# EPICS substitutions: splineApp/Db/transformations.substitutions
file spline.template

{
  pattern{ DEV, LOCA, UNIT, FILENAME }
         { UND, TEST, MC, current}

}
